{attribute addProperty BoxType "EL9576-0000-0022"}
{attribute addProperty Id "BCT_InputsAT %I*BCT_Inputs_4FFA390D136170WcStateAT %I*WcState_F855686C1620InfoDataAT %I*InfoData_BC63D37F80100"}
{attribute addProperty CRC "2937750143"}
{attribute addProperty SizeInBites "232"}
{attribute addProperty SizeInBytes "29"}
TYPE EL9576_B5DF83EF :
STRUCT
	{attribute addProperty Name "BCT_Inputs"}
	BCT_Inputs : BCT_Inputs_4FFA390D;
	{attribute addProperty Name "WcState"}
	WcState : WcState_F855686C;
	{attribute addProperty Name "InfoData"}
	InfoData : InfoData_BC63D37F;
END_STRUCT
END_TYPE

(* stored: Version 1.2.0.0, ProductVersion 3.1.4024.9
   DUT EL9576_B5DF83EF: Id {f8aba60c-5130-42a0-9fed-ff30dcae8a4c} *)
